FUNCTION_BLOCK FB_ExecutorCut EXTENDS FB_ExecutorBase
VAR
	_CutDirection : E_CutDirection; //   0 - Cutter direction X, 1 - Cutter direction Y, you can add more in the Enum
END_VAR

PROPERTY CutDirection : E_CutDirection
GET
CutDirection := _CutDirection;
END_GET
SET
_CutDirection := CutDirection;
END_SET
END_PROPERTY

METHOD PUBLIC CyclicLogic
VAR_INST
    localConfig   : ST_GantryXYZ_Config;
    currentSeg    : ST_CutSegment;
    
    // Ujednolicone zmienne pomocnicze
    totalSegments : INT;
    offsetX       : REAL;
    offsetY       : REAL;
END_VAR

// --- START LOGIKI ---
StepTimer();

IF _RecipeBuilder = 0 OR _ConfigProvider = 0 THEN RETURN; END_IF

localConfig := _ConfigProvider.Config;

// ========================================================
// MAGICZNY ROZDZIELACZ Z ENUMEM
// ========================================================
CASE CutDirection OF
    E_CutDirection.eCutX:
        IF iCurrentSegment < 1 OR iCurrentSegment > 32 THEN iCurrentSegment := 1; END_IF
        currentSeg    := _RecipeBuilder.SegmentsCutX[iCurrentSegment];
        totalSegments := _RecipeBuilder.SegmentsToCutX;
        offsetX       := localConfig.CutterXOffsetX;
        offsetY       := localConfig.CutterXOffsetY;
        
    E_CutDirection.eCutY:
        IF iCurrentSegment < 1 OR iCurrentSegment > 32 THEN iCurrentSegment := 1; END_IF
        currentSeg    := _RecipeBuilder.SegmentsCutY[iCurrentSegment];
        totalSegments := _RecipeBuilder.SegmentsToCutY;
        offsetX       := localConfig.CutterYOffsetX;
        offsetY       := localConfig.CutterYOffsetY;
        
END_CASE
// ========================================================


CASE nStep OF
    0: // IDLE
    
    5: // INIT
        IF _AxisX.Enable() AND _AxisY.Enable() AND _AxisZ.Enable() THEN
            IF totalSegments <= 0 THEN
                nStep := 1000;
                RETURN;
            END_IF;

            _AxisX.Acceleration := 500; _AxisX.Deceleration := 8000;
            _AxisY.Acceleration := 500; _AxisY.Deceleration := 8000;
            _AxisZ.Acceleration := 500; _AxisZ.Deceleration := 8000;
            
            _AxisX.Velocity := localConfig.RapidSpeedX;
            _AxisY.Velocity := localConfig.RapidSpeedY;
            _AxisZ.Velocity := localConfig.RapidSpeedZ;

            iCurrentSegment := 1;
            IF NOT _AxisX.Busy AND NOT _AxisY.Busy AND NOT _AxisZ.Busy THEN nStep := 10; END_IF     
        END_IF

    // -------- Dojazd do początku cięcia --------
    10:
        // Zobacz jak czysto to teraz wygląda! Żadnych X/Y, po prostu używamy zmiennych z rozdzielacza:
        _AxisX.MoveAbsolute(currentSeg.Start.X + offsetX + localConfig.GlobalOffset, 0);
        _AxisY.MoveAbsolute(currentSeg.Start.Y + offsetY + localConfig.GlobalOffset, 0);
        nStep := 20;

    20: // Czekamy na pozycję XY
        IF _AxisX.InPosition AND _AxisY.InPosition THEN nStep := 30;
        ELSIF _AxisX.Error OR _AxisY.Error THEN nStep := 999; END_IF

    30: // Wysunięcie siłownika (obojętnie jakiego, bo to wie interfejs _Cylinder!)
        _Cylinder.Extend();
        nStep := 40;

    40: 
        IF _Cylinder.Extended THEN
            // Bierzemy prędkość cięcia (tu też możemy zrobić małego if'a, jeśli zależy nam na precyzji,
            // bo w starym kodzie zawsze brałeś CuttingSpeedX i Y[cite: 3757, 3758]. Zostawiam obie)
            _AxisX.Velocity := localConfig.CuttingSpeedX;
            _AxisY.Velocity := localConfig.CuttingSpeedY;
            nStep := 50;
        ELSIF _Cylinder.Error THEN nStep := 999; END_IF
            
    50: // Czekanie
        StepTimer(IN := TRUE, PT := REAL_TO_TIME(localConfig.CuttingIdleTime * 1000.0));
        IF StepTimer.Q THEN StepTimer(IN := FALSE); nStep := 60; END_IF

    60: // Cięcie XY do końca
        _AxisX.MoveAbsolute(currentSeg.Stop.X + offsetX + localConfig.GlobalOffset, 0);
        _AxisY.MoveAbsolute(currentSeg.Stop.Y + offsetY + localConfig.GlobalOffset, 0);
        nStep := 70;

    70: // Czekamy na koniec cięcia
        IF _AxisX.InPosition AND _AxisY.InPosition THEN nStep := 80;
        ELSIF _AxisX.Error OR _AxisY.Error THEN nStep := 999; END_IF

    80: // Chowanie ostrza
        _Cylinder.Retract();
        nStep := 85;

    85: 
        IF _Cylinder.Retracted THEN
             iCurrentSegment := iCurrentSegment + 1;
             nStep := 90;
        ELSIF _Cylinder.Error THEN nStep := 999; END_IF    

    90: // Drugi Idle Time
        StepTimer(IN := TRUE, PT := REAL_TO_TIME(localConfig.CuttingIdleTime * 1000.0));
        IF StepTimer.Q THEN
            StepTimer(IN := FALSE);
            _AxisX.Velocity := localConfig.RapidSpeedX;
            _AxisY.Velocity := localConfig.RapidSpeedY;
            
            // Decyzja o powrocie na bazie uniwersalnej zmiennej
            IF iCurrentSegment > totalSegments THEN nStep := 1000;
            ELSE nStep := 10; END_IF
        END_IF

    999: // Błąd
        _bBusy := FALSE; _bError := TRUE; _bDone := FALSE; nStep := 0;

    1000: // Koniec
        _bBusy := FALSE; _bDone := TRUE; nStep := 0;
END_CASE
END_METHOD

END_FUNCTION_BLOCK

(* stored: Version 1.1.0.1, ProductVersion 3.1.4024.15
   POU FB_ExecutorCut: Id {d112f497-12ba-4ef0-9a18-d5d0a0a5cb2a}, SpecialFunc None
   Property CutDirection: Id {2e5b2549-487e-4c71-8ab5-2707083adbce}
   Get Get: Id {78fa6f30-8cfc-4c8f-b630-a087ae846ffd}
   Set Set: Id {a2853fb5-b406-4a3c-b3c2-cbf02554944c}
   Method CyclicLogic: Id {0b527001-8b78-458c-8b6f-271e71aa0862} *)
